% RSLogix 500 project pump_vibration_alarm.RSS, saved by version 8.30.00.16 %
PROJECT "UNTITLED"    % processor: Bul.1763 MicroLogix 1100 Series B %

PROGRAM FILES
  LAD 2 "MAIN"  5 rungs
  LAD 3 "IO"  10 rungs
  LAD 4 "CONTROL"  8 rungs
  LAD 5 "HOA"  7 rungs
  LAD 6 "ALARMS"  9 rungs

DATA FILES
  O0 OUTPUT  4 elements
  I1 INPUT  6 elements
  S2 STATUS  66 elements
  B3 BINARY  4 elements
  T4 TIMER  6 elements
  C5 COUNTER  1 elements
  R6 CONTROL  1 elements
  N7 INTEGER  4 elements
  F8 FLOAT  1 elements

LADDER 2 "MAIN"
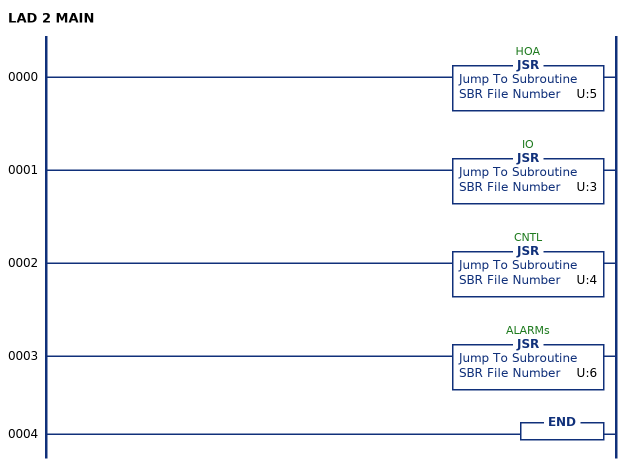
% Rung: 0 %
SOR JSR U:5 EOR
%   U:5  "HOA" %
% Rung: 1 %
SOR JSR U:3 EOR
%   U:3  "IO" %
% Rung: 2 %
SOR JSR U:4 EOR
%   U:4  "CNTL" %
% Rung: 3 %
SOR JSR U:6 EOR
%   U:6  "ALARMs" %
% Rung: 4 %
SOR END EOR

LADDER 3 "IO"
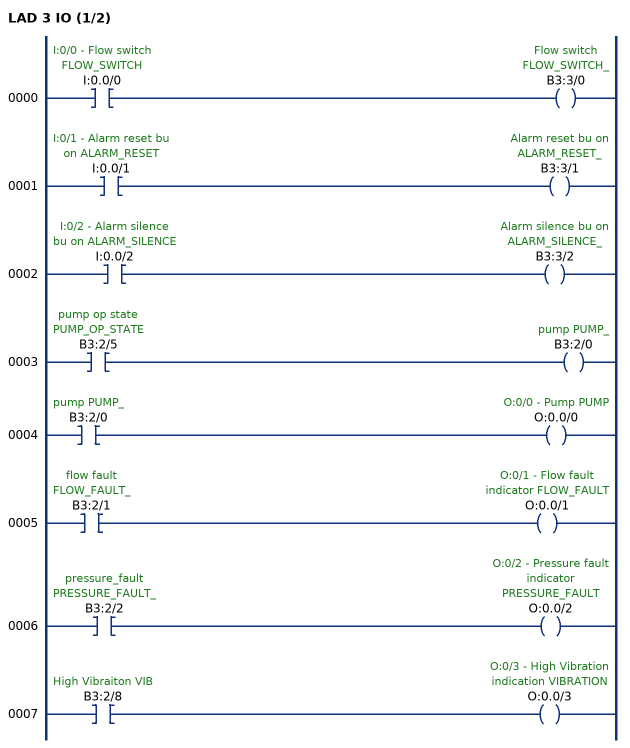
% Rung: 0 %
SOR XIC I:0.0/0 OTE B3:3/0 EOR
%   I:0.0/0  FLOW_SWITCH  "I:0/0 - Flow switch" %
%   B3:3/0  FLOW_SWITCH_  "Flow switch" %
% Rung: 1 %
SOR XIC I:0.0/1 OTE B3:3/1 EOR
%   I:0.0/1  ALARM_RESET  "I:0/1 - Alarm reset bu on" %
%   B3:3/1  ALARM_RESET_  "Alarm reset bu on" %
% Rung: 2 %
SOR XIC I:0.0/2 OTE B3:3/2 EOR
%   I:0.0/2  ALARM_SILENCE  "I:0/2 - Alarm silence bu on" %
%   B3:3/2  ALARM_SILENCE_  "Alarm silence bu on" %
% Rung: 3 %
SOR XIC B3:2/5 OTE B3:2/0 EOR
%   B3:2/5  PUMP_OP_STATE  "pump op state" %
%   B3:2/0  PUMP_  "pump" %
% Rung: 4 %
SOR XIC B3:2/0 OTE O:0.0/0 EOR
%   B3:2/0  PUMP_  "pump" %
%   O:0.0/0  PUMP  "O:0/0 - Pump" %
% Rung: 5 %
SOR XIC B3:2/1 OTE O:0.0/1 EOR
%   B3:2/1  FLOW_FAULT_  "flow fault" %
%   O:0.0/1  FLOW_FAULT  "O:0/1 - Flow fault indicator" %
% Rung: 6 %
SOR XIC B3:2/2 OTE O:0.0/2 EOR
%   B3:2/2  PRESSURE_FAULT_  "pressure_fault" %
%   O:0.0/2  PRESSURE_FAULT  "O:0/2 - Pressure fault indicator" %
% Rung: 7 %
SOR XIC B3:2/8 OTE O:0.0/3 EOR
%   B3:2/8  VIB  "High Vibraiton" %
%   O:0.0/3  VIBRATION  "O:0/3 - High Vibration indication" %

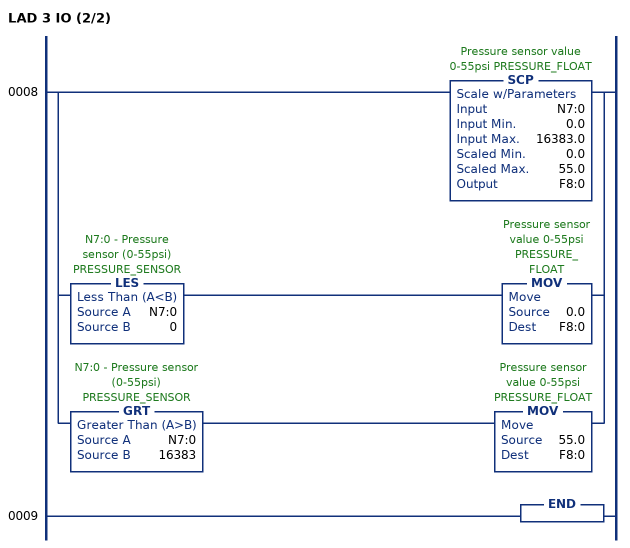
% Rung: 8 %
SOR BST SCP N7:0 0.0 16383.0 0.0 55.0 F8:0 NXB LES N7:0 0 MOV 0.0 F8:0 NXB GRT N7:0 16383 MOV 55.0 F8:0 BND EOR
%   N7:0  PRESSURE_SENSOR  "N7:0 - Pressure sensor (0-55psi)" %
%   F8:0  PRESSURE_FLOAT  "Pressure sensor value 0-55psi" %
% Rung: 9 %
SOR END EOR

LADDER 4 "CONTROL"
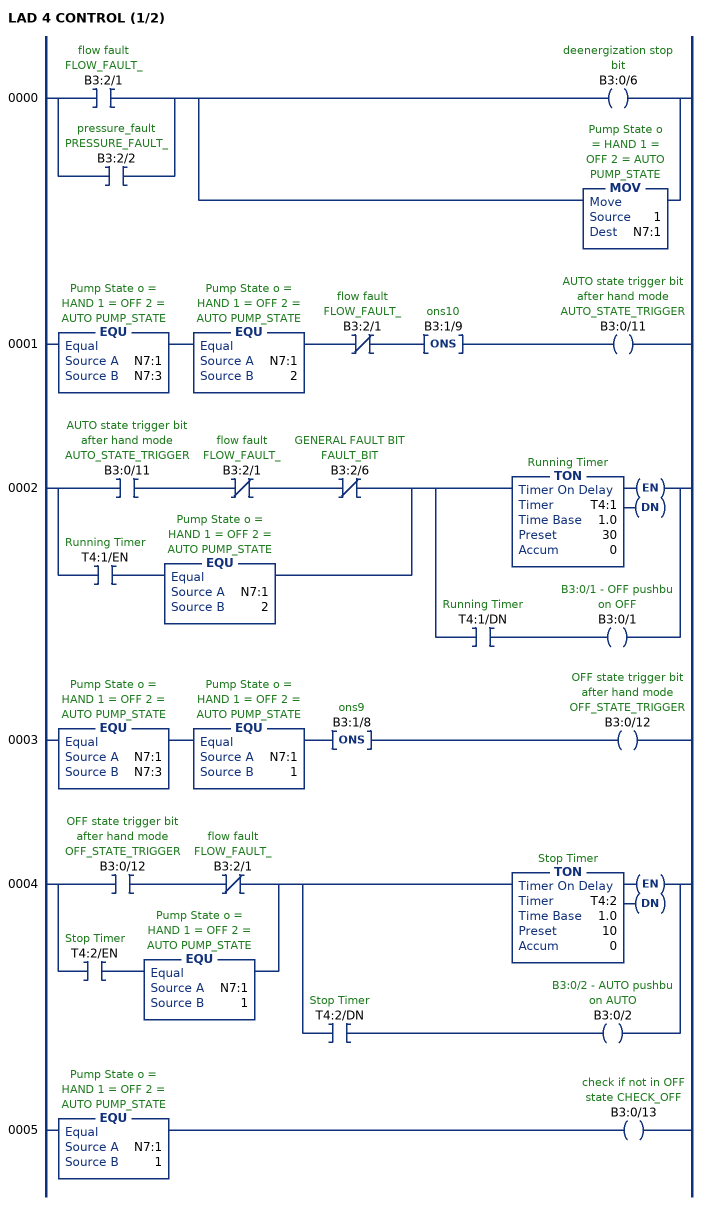
% Rung: 0 %
SOR BST XIC B3:2/1 NXB XIC B3:2/2 BND BST OTE B3:0/6 NXB MOV 1 N7:1 BND EOR
%   B3:2/1  FLOW_FAULT_  "flow fault" %
%   B3:2/2  PRESSURE_FAULT_  "pressure_fault" %
%   B3:0/6  "deenergization stop bit" %
%   N7:1  PUMP_STATE  "Pump State o = HAND 1 = OFF 2 = AUTO" %
% Rung: 1 %
SOR EQU N7:1 N7:3 EQU N7:1 2 XIO B3:2/1 ONS B3:1/9 OTE B3:0/11 EOR
%   N7:1  PUMP_STATE  "Pump State o = HAND 1 = OFF 2 = AUTO" %
%   N7:3  PREVIOUS_STATE  "temporary pump state integer" %
%   B3:2/1  FLOW_FAULT_  "flow fault" %
%   B3:1/9  "ons10" %
%   B3:0/11  AUTO_STATE_TRIGGER  "AUTO state trigger bit after hand mode" %
% Rung: 2 %
SOR BST XIC B3:0/11 XIO B3:2/1 XIO B3:2/6 NXB XIC T4:1/EN EQU N7:1 2 BND BST TON T4:1 1.0 30 0 NXB XIC T4:1/DN OTE B3:0/1 BND EOR
%   B3:0/11  AUTO_STATE_TRIGGER  "AUTO state trigger bit after hand mode" %
%   B3:2/1  FLOW_FAULT_  "flow fault" %
%   B3:2/6  FAULT_BIT  "GENERAL FAULT BIT" %
%   T4:1  "Running Timer" %
%   N7:1  PUMP_STATE  "Pump State o = HAND 1 = OFF 2 = AUTO" %
%   B3:0/1  OFF  "B3:0/1 - OFF pushbu on" %
% Rung: 3 %
SOR EQU N7:1 N7:3 EQU N7:1 1 ONS B3:1/8 OTE B3:0/12 EOR
%   N7:1  PUMP_STATE  "Pump State o = HAND 1 = OFF 2 = AUTO" %
%   N7:3  PREVIOUS_STATE  "temporary pump state integer" %
%   B3:1/8  "ons9" %
%   B3:0/12  OFF_STATE_TRIGGER  "OFF state trigger bit after hand mode" %
% Rung: 4 %
SOR BST XIC B3:0/12 XIO B3:2/1 NXB XIC T4:2/EN EQU N7:1 1 BND BST TON T4:2 1.0 10 0 NXB XIC T4:2/DN OTE B3:0/2 BND EOR
%   B3:0/12  OFF_STATE_TRIGGER  "OFF state trigger bit after hand mode" %
%   B3:2/1  FLOW_FAULT_  "flow fault" %
%   T4:2  "Stop Timer" %
%   N7:1  PUMP_STATE  "Pump State o = HAND 1 = OFF 2 = AUTO" %
%   B3:0/2  AUTO  "B3:0/2 - AUTO pushbu on" %
% Rung: 5 %
SOR EQU N7:1 1 OTE B3:0/13 EOR
%   N7:1  PUMP_STATE  "Pump State o = HAND 1 = OFF 2 = AUTO" %
%   B3:0/13  CHECK_OFF  "check if not in OFF state" %

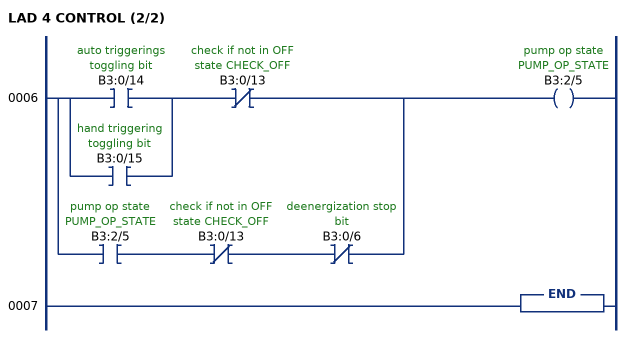
% Rung: 6 %
SOR BST BST XIC B3:0/14 NXB XIC B3:0/15 BND XIO B3:0/13 NXB XIC B3:2/5 XIO B3:0/13 XIO B3:0/6 BND OTE B3:2/5 EOR
%   B3:0/14  "auto triggerings toggling bit" %
%   B3:0/15  "hand triggering toggling bit" %
%   B3:0/13  CHECK_OFF  "check if not in OFF state" %
%   B3:2/5  PUMP_OP_STATE  "pump op state" %
%   B3:0/6  "deenergization stop bit" %
% Rung: 7 %
SOR END EOR

LADDER 5 "HOA"
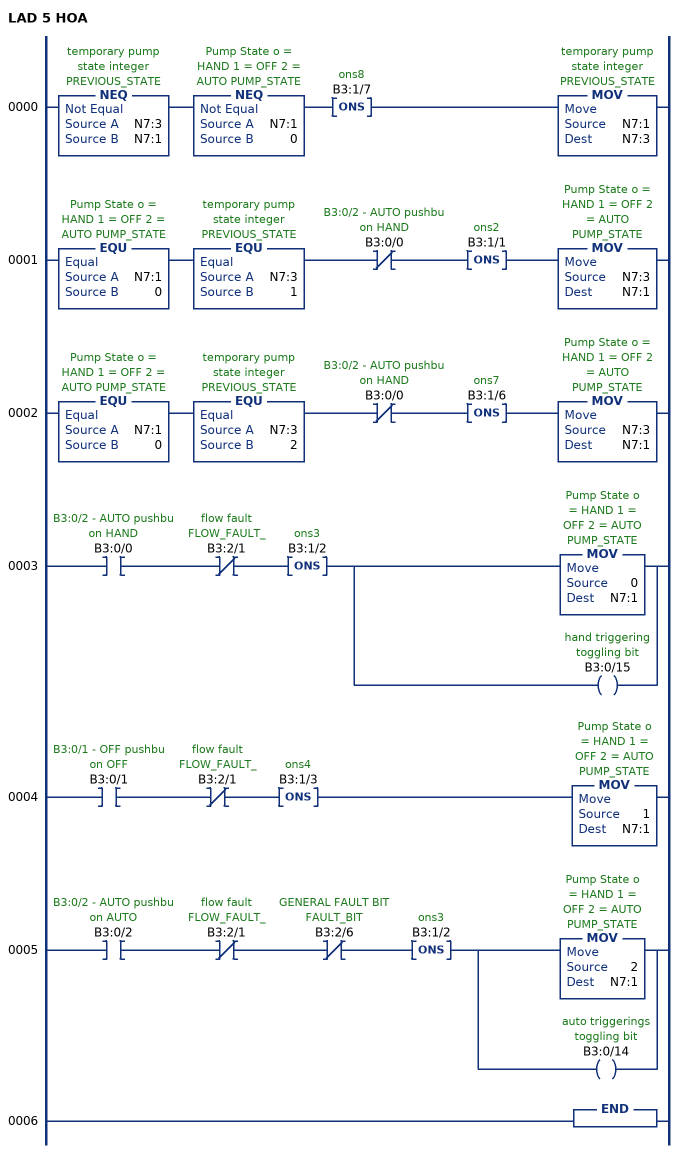
% Rung: 0 %
SOR NEQ N7:3 N7:1 NEQ N7:1 0 ONS B3:1/7 MOV N7:1 N7:3 EOR
%   N7:3  PREVIOUS_STATE  "temporary pump state integer" %
%   N7:1  PUMP_STATE  "Pump State o = HAND 1 = OFF 2 = AUTO" %
%   B3:1/7  "ons8" %
% Rung: 1 %
SOR EQU N7:1 0 EQU N7:3 1 XIO B3:0/0 ONS B3:1/1 MOV N7:3 N7:1 EOR
%   N7:1  PUMP_STATE  "Pump State o = HAND 1 = OFF 2 = AUTO" %
%   N7:3  PREVIOUS_STATE  "temporary pump state integer" %
%   B3:0/0  HAND  "B3:0/2 - AUTO pushbu on" %
%   B3:1/1  "ons2" %
% Rung: 2 %
SOR EQU N7:1 0 EQU N7:3 2 XIO B3:0/0 ONS B3:1/6 MOV N7:3 N7:1 EOR
%   N7:1  PUMP_STATE  "Pump State o = HAND 1 = OFF 2 = AUTO" %
%   N7:3  PREVIOUS_STATE  "temporary pump state integer" %
%   B3:0/0  HAND  "B3:0/2 - AUTO pushbu on" %
%   B3:1/6  "ons7" %
% Rung: 3 %
SOR XIC B3:0/0 XIO B3:2/1 ONS B3:1/2 BST MOV 0 N7:1 NXB OTE B3:0/15 BND EOR
%   B3:0/0  HAND  "B3:0/2 - AUTO pushbu on" %
%   B3:2/1  FLOW_FAULT_  "flow fault" %
%   B3:1/2  "ons3" %
%   N7:1  PUMP_STATE  "Pump State o = HAND 1 = OFF 2 = AUTO" %
%   B3:0/15  "hand triggering toggling bit" %
% Rung: 4 %
SOR XIC B3:0/1 XIO B3:2/1 ONS B3:1/3 MOV 1 N7:1 EOR
%   B3:0/1  OFF  "B3:0/1 - OFF pushbu on" %
%   B3:2/1  FLOW_FAULT_  "flow fault" %
%   B3:1/3  "ons4" %
%   N7:1  PUMP_STATE  "Pump State o = HAND 1 = OFF 2 = AUTO" %
% Rung: 5 %
SOR XIC B3:0/2 XIO B3:2/1 XIO B3:2/6 ONS B3:1/2 BST MOV 2 N7:1 NXB OTE B3:0/14 BND EOR
%   B3:0/2  AUTO  "B3:0/2 - AUTO pushbu on" %
%   B3:2/1  FLOW_FAULT_  "flow fault" %
%   B3:2/6  FAULT_BIT  "GENERAL FAULT BIT" %
%   B3:1/2  "ons3" %
%   N7:1  PUMP_STATE  "Pump State o = HAND 1 = OFF 2 = AUTO" %
%   B3:0/14  "auto triggerings toggling bit" %
% Rung: 6 %
SOR END EOR

LADDER 6 "ALARMS"
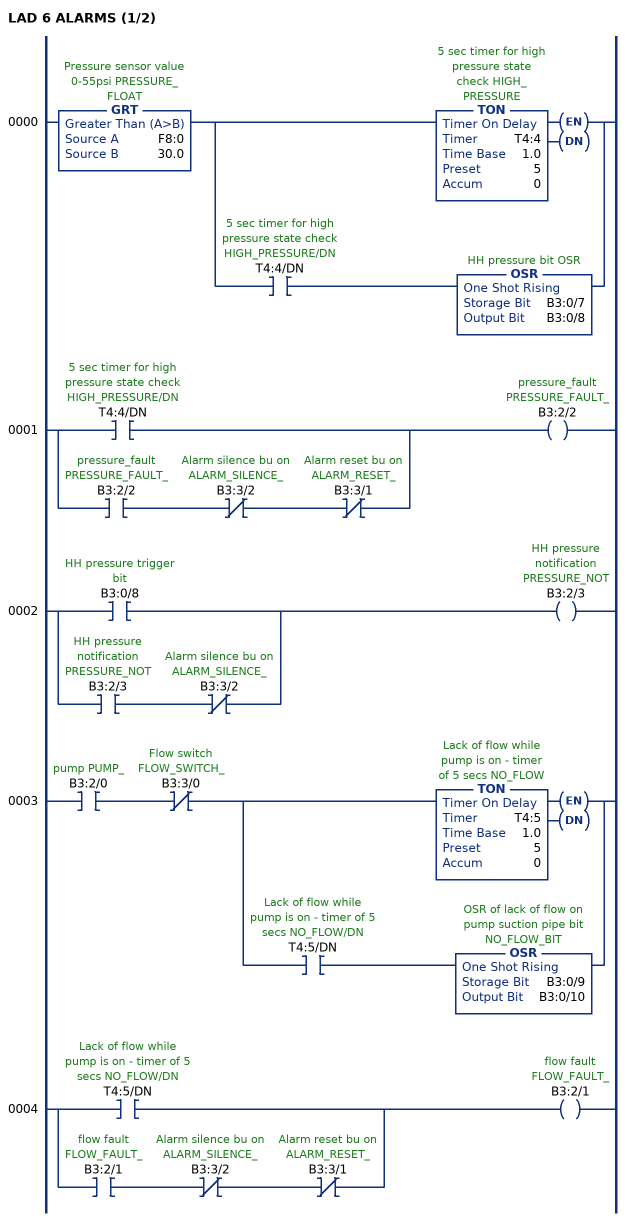
% Rung: 0 %
SOR GRT F8:0 30.0 BST TON T4:4 1.0 5 0 NXB XIC T4:4/DN OSR B3:0/7 B3:0/8 BND EOR
%   F8:0  PRESSURE_FLOAT  "Pressure sensor value 0-55psi" %
%   T4:4  HIGH_PRESSURE  "5 sec timer for high pressure state check" %
%   B3:0/7  "HH pressure bit OSR" %
%   B3:0/8  "HH pressure trigger bit" %
% Rung: 1 %
SOR BST XIC T4:4/DN NXB XIC B3:2/2 XIO B3:3/2 XIO B3:3/1 BND OTE B3:2/2 EOR
%   T4:4  HIGH_PRESSURE  "5 sec timer for high pressure state check" %
%   B3:2/2  PRESSURE_FAULT_  "pressure_fault" %
%   B3:3/2  ALARM_SILENCE_  "Alarm silence bu on" %
%   B3:3/1  ALARM_RESET_  "Alarm reset bu on" %
% Rung: 2 %
SOR BST XIC B3:0/8 NXB XIC B3:2/3 XIO B3:3/2 BND OTE B3:2/3 EOR
%   B3:0/8  "HH pressure trigger bit" %
%   B3:2/3  PRESSURE_NOT  "HH pressure notification" %
%   B3:3/2  ALARM_SILENCE_  "Alarm silence bu on" %
% Rung: 3 %
SOR XIC B3:2/0 XIO B3:3/0 BST TON T4:5 1.0 5 0 NXB XIC T4:5/DN OSR B3:0/9 B3:0/10 BND EOR
%   B3:2/0  PUMP_  "pump" %
%   B3:3/0  FLOW_SWITCH_  "Flow switch" %
%   T4:5  NO_FLOW  "Lack of flow while pump is on - timer of 5 secs" %
%   B3:0/9  NO_FLOW_BIT  "OSR of lack of flow on pump suction pipe bit" %
%   B3:0/10  "lack of flow trigger bit OSR" %
% Rung: 4 %
SOR BST XIC T4:5/DN NXB XIC B3:2/1 XIO B3:3/2 XIO B3:3/1 BND OTE B3:2/1 EOR
%   T4:5  NO_FLOW  "Lack of flow while pump is on - timer of 5 secs" %
%   B3:2/1  FLOW_FAULT_  "flow fault" %
%   B3:3/2  ALARM_SILENCE_  "Alarm silence bu on" %
%   B3:3/1  ALARM_RESET_  "Alarm reset bu on" %

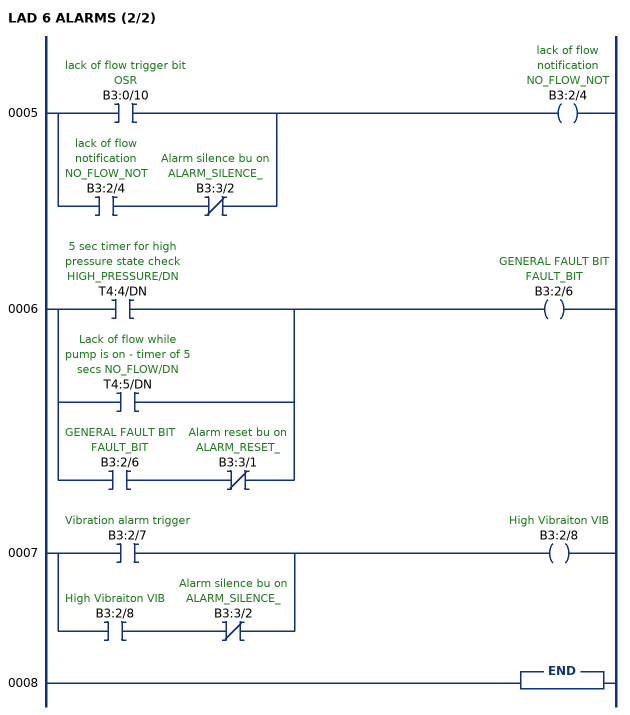
% Rung: 5 %
SOR BST XIC B3:0/10 NXB XIC B3:2/4 XIO B3:3/2 BND OTE B3:2/4 EOR
%   B3:0/10  "lack of flow trigger bit OSR" %
%   B3:2/4  NO_FLOW_NOT  "lack of flow notification" %
%   B3:3/2  ALARM_SILENCE_  "Alarm silence bu on" %
% Rung: 6 %
SOR BST BST XIC T4:4/DN NXB XIC T4:5/DN BND NXB XIC B3:2/6 XIO B3:3/1 BND OTE B3:2/6 EOR
%   T4:4  HIGH_PRESSURE  "5 sec timer for high pressure state check" %
%   T4:5  NO_FLOW  "Lack of flow while pump is on - timer of 5 secs" %
%   B3:2/6  FAULT_BIT  "GENERAL FAULT BIT" %
%   B3:3/1  ALARM_RESET_  "Alarm reset bu on" %
% Rung: 7 %
SOR BST XIC B3:2/7 NXB XIC B3:2/8 XIO B3:3/2 BND OTE B3:2/8 EOR
%   B3:2/7  "Vibration alarm trigger" %
%   B3:2/8  VIB  "High Vibraiton" %
%   B3:3/2  ALARM_SILENCE_  "Alarm silence bu on" %
% Rung: 8 %
SOR END EOR

OTHER DOCUMENTED ADDRESSES
  B3:0/3  "First pass triggering"
  B3:0/4  PUMP_TRIGGER  "pump run triggering"
  B3:0/5  FLOW_CHECK_BIT  "5secs flow check bit"
  B3:1/0  "ons1"
  B3:1/4  "ons5"
  B3:1/5  "ons6"
  B3:1/10  "ons11"
  N7:2  PRESSURE  "N7:0 - Pressure sensor (0-55psi)"
  T4:3  "Flow detection timer"

DATA TABLE (non-zero values as saved)
DATA T4
% .PRE .ACC %
% T4:1 % 30 0
% T4:2 % 10 0
% T4:3 % 5 0
% T4:4 % 5 0
% T4:5 % 5 0
DATA N7
% N7:0 % 8192 0 0 0
